Yaskawa INFORM job: R1_W27-A5(90,0)OK-KM.JBI

/JOB
//NAME R1_W27-A5(90,0)OK-KM
///FOLDERNAME KRIS-SCIANA
//POS
///NPOS 185,185,0,11,0,0
///TOOL 0
///POSTYPE PULSE
///PULSE
C00000=37728,-25402,-59646,12123,81500,-87547
C00001=37728,-25402,-59646,12123,81500,-87547
C00002=91138,-155068,-109614,11761,-43738,-37693
C00003=119745,-153431,-102899,11459,-45100,-35884
C00004=119745,-153431,-102899,-27163,23845,-36063
C00005=82911,-33235,-23976,-38303,40316,-52135
C00006=76873,-23146,-17071,-33335,38547,-55116
C00007=77767,-16866,-4062,-37722,34988,-52633
C00008=77963,-15290,-967,-38851,34204,-52007
C00009=77963,-14962,-89,-39196,33912,-51822
C00010=77963,-15290,-967,-38851,34204,-52007
C00011=74912,-28085,-18084,-33157,36163,-55249
C00012=87425,-27898,-13680,-43892,39692,-48702
C00013=86506,-25121,-9781,-44194,38523,-48572
C00014=85850,-24209,-8487,-44098,37958,-48664
C00015=86506,-25121,-9781,-44194,38523,-48572
C00016=88499,-29485,-18641,-42732,41870,-49349
C00017=84065,-39934,-28269,-47565,31902,-47281
C00018=97660,-57598,-46315,-76057,51112,-44177
C00019=97660,-57598,-46315,-76057,51112,22687
C00020=84258,-1988,-20698,-34156,82686,37449
C00021=71650,44734,31864,-29990,67100,37520
C00022=68559,51841,34481,-21650,72595,35300
C00023=68559,52177,36557,-21773,71566,35494
C00024=71650,44734,31864,-29990,67100,37520
C00025=70945,44192,31290,-29757,66915,37278
C00026=71650,44734,31864,-29990,67100,37520
C00027=73638,27072,10407,-29859,71409,37151
C00028=84818,-5861,-34609,-25685,107970,66305
C00029=82304,-18126,-38436,-25115,103648,66333
C00030=82304,-18241,-37568,-25043,103108,66450
C00031=82304,-18126,-38436,-25115,103648,66333
C00032=81928,-19595,-39516,-25102,103455,66234
C00033=82304,-18126,-38436,-25115,103648,66333
C00034=89590,-10169,-38886,-25731,109749,67700
C00035=79821,25746,-12201,-14172,109985,-51685
C00036=75346,32608,-5411,-14115,108620,-53087
C00037=69367,42381,13672,-2650,109038,-53623
C00038=69672,41657,12911,-2619,109144,-53518
C00039=69367,42407,13451,-2654,109187,-53626
C00040=69778,41548,11559,-2621,109922,-53494
C00041=69778,41458,12200,-2614,109483,-53485
C00042=69778,41717,10519,-2636,110650,-53511
C00043=75546,32003,-7767,-2128,117063,-51505
C00044=89590,-10367,-38270,-25645,109314,67802
C00045=81318,-16645,-42899,-25578,106543,65314
C00046=81011,-17824,-43775,-25562,106392,65231
C00047=81318,-16645,-42899,-25578,106543,65314
C00048=81318,-16217,-44241,-25738,107491,65096
C00049=80508,-19487,-45963,-25627,106690,64976
C00050=80508,-19653,-45420,-25564,106310,65064
C00051=80508,-19487,-45963,-25627,106690,64976
C00052=95846,-36399,-54281,-36372,102338,70376
C00053=102769,-67405,-57032,-50388,80798,81585
C00054=102006,-67104,-56883,-50326,80418,81392
C00055=101071,-66717,-56691,-50243,79954,81156
C00056=102358,-67245,-56953,-50356,80595,81483
C00057=109446,-46040,-50390,-50619,88983,80633
C00058=76818,2269,-30427,-25766,107073,87842
C00059=74377,-18,-31232,-25562,105749,87240
C00060=73964,56,-31169,-25544,105627,87112
C00061=74377,-18,-31232,-25562,105749,87240
C00062=74377,525,-32636,-25731,106781,87003
C00063=73295,1251,-31494,-25627,106170,86744
C00064=73295,967,-30757,-25541,105628,86868
C00065=73295,1251,-31494,-25627,106170,86744
C00066=70279,40415,5647,-25108,102815,86384
C00067=70279,40232,6317,-25050,102354,86487
C00068=70279,40415,5647,-25108,102815,86384
C00069=71244,41386,6665,-25146,102979,86705
C00070=70901,41880,8462,-25047,102103,86769
C00071=70442,41953,8538,-25022,101961,86631
C00072=70902,41930,8262,-25048,102238,86740
C00073=61610,48110,15922,-22399,84700,84261
C00074=61413,48286,16169,-22315,84306,84210
C00075=61008,48239,16118,-22214,84206,84086
C00076=61413,48286,16169,-22315,84306,84210
C00077=61413,48513,15025,-22296,85069,84067
C00078=60697,48720,15417,-22121,84760,83876
C00079=60697,48582,16098,-22134,84306,83960
C00080=60697,48720,15417,-22121,84760,83876
C00081=63518,20060,-6225,-30680,67231,85063
C00082=64098,14214,-10771,-32409,63712,85286
C00083=68885,5587,-7565,-48592,41009,78461
C00084=65627,18359,4931,-47317,38515,77893
C00085=65380,18933,5464,-47167,38362,77820
C00086=65627,18359,4931,-47317,38515,77893
C00087=65627,18423,5468,-47595,38308,78054
C00088=65627,18359,4931,-47317,38515,77893
C00089=70388,-714,-11888,-50078,41438,79261
C00090=70090,148,-11169,-50028,41395,-62740
C00091=64431,-8095,-22559,-54079,48047,-56053
C00092=60138,2499,-10245,-53390,44291,-56175
C00093=60864,4119,-8811,-53841,44675,-55941
C00094=50454,6570,-14378,-8272,39887,-77071
C00095=46890,10124,-11410,8335,39857,-85304
C00096=49558,3708,-17404,-7293,40191,-77557
C00097=52170,-20958,-36880,-10077,39785,-76177
C00098=53236,-23702,-38850,-11204,39728,-75616
C00099=68411,-25809,-57189,-29389,70593,82687
C00100=64998,-21965,-41730,-29205,62846,83456
C00101=47332,3816,-28668,-14363,85152,86760
C00102=13605,-12882,-44436,-5505,92305,85655
C00103=22082,-48383,-67711,-6096,86634,88967
C00104=44284,-41688,-65263,-13455,83816,85908
C00105=48658,1110,-32244,-14746,86156,87078
C00106=44206,2405,-29873,-10094,85398,89089
C00107=46271,27497,-4271,-10640,75407,89194
C00108=49813,9574,-21485,-13963,73922,89293
C00109=51221,-59455,-73476,-13519,71647,80934
C00110=20614,-34885,-59650,-13331,96803,87930
C00111=10167,-61122,-75524,-13198,98224,81006
C00112=18568,-72268,-87151,-10294,92386,67226
C00113=26792,-77751,-90608,-11605,92779,-33394
C00114=45042,-57080,-44270,-29328,87501,-26999
C00115=29931,-98809,-62657,-30113,73342,-29188
C00116=11116,-94328,-56612,-18416,63270,-35426
C00117=11737,-97137,-54513,-22781,52265,-32783
C00118=45210,-102279,-54102,-43605,63453,-17867
C00119=65059,-108164,-59991,-34964,63220,70148
C00120=52273,-70600,-39377,-24696,79942,57751
C00121=43673,-95736,-42893,-26460,67675,57325
C00122=28563,-66776,-31973,-25457,70564,50966
C00123=34229,-67024,-36548,-25195,74692,52186
C00124=29998,-46574,-23957,-5282,52394,19779
C00125=26910,-15086,7402,-4123,49104,18623
C00126=30725,5348,23556,-5801,49891,20233
C00127=26399,10546,29797,6839,45413,17161
C00128=25240,116,19359,9501,43500,14765
C00129=22231,-28513,-5139,11190,44238,13411
C00130=78144,-23782,-17517,-19802,53604,-33534
C00131=71297,46402,29834,-2695,101694,-44274
C00132=54466,25430,16217,2924,106693,-49878
C00133=60216,41298,32233,4120,104740,-47883
C00134=58235,32090,17782,3799,108986,-48454
C00135=79593,-22722,-23344,-19568,57852,-33734
C00136=78528,-18616,-11242,-20296,52560,-33151
C00137=78932,-16743,-10167,-20417,52946,-33052
C00138=78544,-16737,-8595,-20480,51941,-33014
C00139=77955,-18452,-11115,-20012,52425,-33380
C00140=78575,-16130,-9486,-20269,52757,-33170
C00141=76564,-15411,-8500,-18566,50879,-33728
C00142=75844,-13833,-7410,-18312,50740,-34021
C00143=76952,-15561,-8970,-19469,52340,-33810
C00144=76532,-19770,-12086,-19320,52008,-33932
C00145=90733,-10813,-5342,-38854,64320,-29793
C00146=90042,-7330,-2603,-38655,64092,-30029
C00147=89654,-5763,-1731,-38480,64131,-30226
C00148=90645,-6898,-2268,-38798,64375,-29857
C00149=90264,-6063,-535,-38894,63701,-29768
C00150=89843,-4938,-962,-38544,64174,-30154
C00151=90707,-2014,1381,-38736,64612,-29923
C00152=91454,1636,4460,-38922,64932,-29697
C00153=91128,-2551,1262,-38897,64640,-29735
C00154=91822,-6037,-1569,-39075,64914,-29517
C00155=89351,12292,-5617,-20131,79037,60764
C00156=89352,16382,17787,-21350,67492,62811
C00157=87694,16715,18095,-20947,67047,62250
C00158=87033,16875,18243,-20783,66871,62026
C00159=87546,18694,19932,-20926,66903,62219
C00160=87127,16733,16861,-20697,67624,61924
C00161=86853,17243,18585,-20744,66809,61967
C00162=87778,19395,20596,-20991,66917,62307
C00163=93870,634,-11523,-21410,77965,27109
C00164=93832,30424,31287,-31485,89224,-4964
C00165=93834,30423,31286,-31485,89224,-4963
C00166=93835,30423,31286,-31485,89225,-4963
C00167=93885,30318,29928,-31492,89915,-5134
C00168=93558,28166,29049,-31504,89308,-5095
C00169=93835,30423,31286,-31484,89222,-4963
C00170=93835,30427,31290,-31485,89224,-4963
C00171=93832,30428,31291,-31485,89223,-4964
C00172=78422,20921,22036,-838,76825,9185
C00173=78437,23453,23148,-839,77442,9187
C00174=77317,26936,27718,2138,78128,8741
C00175=79840,22908,23920,-1007,76703,9676
C00176=79114,23558,23278,-919,77424,9420
C00177=78338,19571,8789,758,86105,8103
C00178=114533,-1412,-14551,-12904,94461,10066
C00179=113047,-133639,-110380,-13907,-12366,10665
C00180=113047,-161651,-128625,-13333,-12898,10403
C00181=3699,-161651,-128625,-13333,-12898,10403
C00182=3699,-161651,-128625,-13333,-12898,-84221
C00183=-5596,-96163,-97527,-5645,15530,-80546
C00184=-5408,65526,-18493,9932,83824,-70089
BC00000=244758,1245750,1068204
BC00001=244758,1188259,1068204
BC00002=328514,1188626,1057284
BC00003=25914,1188837,1050998
BC00004=25914,1188837,250553
BC00005=876,1188837,301895
BC00006=876,1188837,280170
BC00007=876,1188837,280170
BC00008=876,1188837,280170
BC00009=876,1188837,280170
BC00010=876,1188837,280170
BC00011=876,1188837,280170
BC00012=876,1188837,280170
BC00013=876,1188837,280170
BC00014=876,1188837,280170
BC00015=876,1188837,280170
BC00016=876,1188837,280170
BC00017=876,1188837,242031
BC00018=876,1188837,199876
BC00019=876,1188837,199876
BC00020=876,1188837,199876
BC00021=876,1188837,199876
BC00022=876,1188837,199876
BC00023=876,1188837,199876
BC00024=876,1188837,199876
BC00025=876,1188837,199873
BC00026=876,1188837,199876
BC00027=876,1188837,199876
BC00028=876,1188837,199876
BC00029=876,1188837,199876
BC00030=876,1188837,199876
BC00031=876,1188837,199876
BC00032=876,1188837,199876
BC00033=876,1188837,199876
BC00034=876,1188837,199876
BC00035=876,1188837,199876
BC00036=876,1188837,199876
BC00037=876,1188837,199876
BC00038=876,1188837,199876
BC00039=876,1188837,199876
BC00040=876,1188837,199876
BC00041=876,1188837,199876
BC00042=876,1188837,199876
BC00043=876,1188837,200133
BC00044=876,1188837,583866
BC00045=876,1188837,583866
BC00046=876,1188837,583866
BC00047=876,1188837,583866
BC00048=876,1188837,583866
BC00049=876,1188837,583866
BC00050=876,1188837,583866
BC00051=876,1188837,583866
BC00052=876,1188837,583866
BC00053=876,1188837,597308
BC00054=876,1188837,597308
BC00055=876,1188837,597308
BC00056=876,1188837,597308
BC00057=876,1188837,597308
BC00058=876,1188837,587630
BC00059=876,1188837,587630
BC00060=876,1188837,587630
BC00061=876,1188837,587630
BC00062=876,1188837,587630
BC00063=876,1188837,587630
BC00064=876,1188837,587630
BC00065=876,1188837,587630
BC00066=876,1188837,587630
BC00067=876,1188837,587630
BC00068=876,1188837,587630
BC00069=876,1188837,587630
BC00070=876,1188837,587628
BC00071=876,1188837,587628
BC00072=876,1188837,587630
BC00073=876,1156999,587630
BC00074=876,1156326,587630
BC00075=876,1156326,587630
BC00076=876,1156326,587630
BC00077=876,1156326,587630
BC00078=876,1156326,587630
BC00079=876,1156326,587630
BC00080=876,1156326,587630
BC00081=876,1156326,587630
BC00082=876,1156326,597308
BC00083=876,1156326,697181
BC00084=876,1156326,697181
BC00085=876,1156326,697181
BC00086=876,1156326,697181
BC00087=876,1156326,697181
BC00088=876,1156326,697181
BC00089=876,1156326,697181
BC00090=876,1156326,697181
BC00091=876,1128921,697181
BC00092=876,1128921,697181
BC00093=876,1128921,697181
BC00094=876,1128921,697181
BC00095=876,1128922,697179
BC00096=876,1128921,697181
BC00097=876,1128921,697181
BC00098=876,1128921,697181
BC00099=1315,1138846,645939
BC00100=1315,1138846,645939
BC00101=1732,1122257,597308
BC00102=2782,1039755,587713
BC00103=2792,1082515,587630
BC00104=1732,1122257,587630
BC00105=1732,1122257,587630
BC00106=1732,1122257,587630
BC00107=1732,1122257,587630
BC00108=1732,1122257,587630
BC00109=1732,1122257,587630
BC00110=1732,1065745,587630
BC00111=1732,1065745,587630
BC00112=1732,1065745,587630
BC00113=1732,1065745,597308
BC00114=1732,1065745,805135
BC00115=1732,1066766,805135
BC00116=1732,1066766,791693
BC00117=1732,1066766,791693
BC00118=1732,1066766,805135
BC00119=1732,1066766,805135
BC00120=1732,1066766,417253
BC00121=29114,1066766,417253
BC00122=5096,1066766,417253
BC00123=1732,1066766,417253
BC00124=1732,1066766,417253
BC00125=1732,1066766,417253
BC00126=1732,1066766,417253
BC00127=1732,1066766,417253
BC00128=1732,1066766,417253
BC00129=1732,1066766,417253
BC00130=876,1188837,310651
BC00131=876,1188837,310651
BC00132=876,1149728,310651
BC00133=876,1149728,310651
BC00134=876,1149728,310651
BC00135=876,1384690,305516
BC00136=876,1384690,305516
BC00137=876,1384690,297010
BC00138=876,1384690,297010
BC00139=876,1384690,297010
BC00140=876,1384690,297005
BC00141=876,1384690,296893
BC00142=876,1384690,296887
BC00143=876,1384690,305393
BC00144=876,1384690,326658
BC00145=876,1384690,316977
BC00146=876,1384690,294261
BC00147=876,1384690,285175
BC00148=876,1384690,285175
BC00149=876,1384690,285175
BC00150=876,1384690,285189
BC00151=876,1384690,285231
BC00152=876,1384690,285245
BC00153=876,1384690,294331
BC00154=876,1384690,317047
BC00155=876,1384690,372171
BC00156=876,1384690,372171
BC00157=876,1384690,350251
BC00158=876,1384690,341483
BC00159=876,1384690,341483
BC00160=876,1384690,341483
BC00161=876,1384690,341468
BC00162=876,1384690,372038
BC00163=876,1384690,372038
BC00164=6218,1373517,366370
BC00165=10148,1372468,343278
BC00166=11720,1372049,334041
BC00167=11720,1372049,334041
BC00168=11720,1372049,334041
BC00169=12357,1372055,334027
BC00170=15563,1372482,343131
BC00171=11633,1373530,366223
BC00172=7822,1384690,403141
BC00173=10818,1384690,380007
BC00174=12016,1384690,370753
BC00175=12016,1384690,370753
BC00176=12016,1384690,370753
BC00177=10869,1187534,355175
BC00178=877,1178820,383119
BC00179=877,1178820,1012132
BC00180=877,1178820,1012132
BC00181=125475,1178820,1012132
BC00182=354926,1178820,1012132
BC00183=329290,1178681,1025649
BC00184=165568,1305468,1058537
///POSTYPE BASE
///RECTAN
///RCONF 0,0,0,0,0,0,0,0,0,0,0,0,0,0,0,0,0,0,0,0,0,0,0,0
P00006=0.222,-3.123,-1.508,0.0000,0.0000,0.0000
P00022=0.222,-3.123,-1.508,0.0000,0.0000,0.0000
P00023=0.143,-0.036,0.682,0.0000,0.0000,0.0000
P00024=0.145,-0.552,1.326,0.0000,0.0000,0.0000
P00025=-2.003,0.006,0.728,0.0000,0.0000,0.0000
P00026=0.562,-0.002,-0.337,0.0000,0.0000,0.0000
P00027=-0.746,0.015,-9.096,0.0000,0.0000,0.0000
P00028=-2.237,-0.018,-7.702,0.0000,0.0000,0.0000
P00029=-2.156,-0.086,-4.681,0.0000,0.0000,0.0000
P00030=5.926,-4.294,-1.390,0.0000,0.0000,0.0000
P00035=2.817,0.591,-1.622,0.0000,0.0000,0.0000
//INST
///DATE 2024/07/29 21:04
///ATTR SC,RW
///GROUP1 RB1,BS1
NOP
SFTOF
MOVJ C00000 BC00000 VJ=50.00
MOVJ C00001 BC00001 VJ=100.00
MOVJ C00002 BC00002 VJ=100.00
MOVJ C00003 BC00003 VJ=100.00
MOVJ C00004 BC00004 VJ=100.00
MOVL C00005 BC00005 V=166.7
MOVL C00006 BC00006 V=166.7
MOVL C00007 BC00007 V=100.0
MOVL C00008 BC00008 V=60.0
REFP 3 C00009 BC00009
CALL JOB:SEARCH-R1
SET P028 P006
SFTON P028
MOVL C00010 BC00010 V=60.0
MOVL C00011 BC00011 V=133.3
MOVL C00012 BC00012 V=133.3
MOVL C00013 BC00013 V=60.0
REFP 3 C00014 BC00014
CALL JOB:SEARCH-R1
SET P028 P006
SFTON P028
MOVL C00015 BC00015 V=60.0
MOVL C00016 BC00016 V=133.3
MOVL C00017 BC00017 V=166.7
'Path S1011
SFTOF
'Path VIA1114
SFTOF
MOVJ C00018 BC00018 VJ=100.00
MOVJ C00019 BC00019 VJ=100.00
'POMIAR NOWE SPOINY
MOVJ C00020 BC00020 VJ=100.00
MOVJ C00021 BC00021 VJ=15.00
MOVL C00022 BC00022 V=83.3
REFP 3 C00023 BC00023
CALL JOB:SEARCH-R1
SET P022 P006
SFTON P022
MOVL C00024 BC00024 V=60.0
REFP 3 C00025 BC00025
CALL JOB:SEARCH-R1
SET P022 P006
SFTON P022
MOVL C00026 BC00026 V=60.0
SFTOF
MOVL C00027 BC00027 V=83.3
MOVL C00028 BC00028 V=83.3
MOVL C00029 BC00029 V=166.7
REFP 3 C00030 BC00030
CALL JOB:SEARCH-R1
SET P023 P006
SFTON P023
MOVL C00031 BC00031 V=60.0
REFP 3 C00032 BC00032
CALL JOB:SEARCH-R1
SET P023 P006
SFTON P023
MOVL C00033 BC00033 V=60.0
MOVJ C00034 BC00034 VJ=15.00
MOVJ C00035 BC00035 VJ=15.00
SFTOF
MOVJ C00036 BC00036 VJ=15.00
'POPRAWIC POMIAR
MOVJ C00037 BC00037 VJ=15.00
REFP 3 C00038 BC00038
CALL JOB:SEARCH-R1
SET P030 P006
SFTON P030
MOVL C00039 BC00039 V=60.0
MOVL C00040 BC00040 V=166.7
REFP 3 C00041 BC00041
CALL JOB:SEARCH-R1
SET P030 P006
SFTON P030
MOVL C00042 BC00042 V=100.0
MOVJ C00043 BC00043 VJ=15.00
SFTOF
MOVJ C00044 BC00044 VJ=50.00
MOVJ C00045 BC00045 VJ=15.00
REFP 3 C00046 BC00046
CALL JOB:SEARCH-R1
SET P024 P006
SFTON P024
MOVL C00047 BC00047 V=60.0
MOVL C00048 BC00048 V=166.7
MOVL C00049 BC00049 V=166.7
REFP 3 C00050 BC00050
CALL JOB:SEARCH-R1
SET P024 P006
SFTON P024
MOVL C00051 BC00051 V=60.0
MOVJ C00052 BC00052 VJ=15.00
SFTOF
MOVJ C00053 BC00053 VJ=15.00
MOVL C00054 BC00054 V=83.3
REFP 3 C00055 BC00055
CALL JOB:SEARCH-R1
SET P024 P006
SFTON P024
MOVL C00056 BC00056 V=83.3
MOVL C00057 BC00057 V=833.3
MOVJ C00058 BC00058 VJ=15.00
MOVL C00059 BC00059 V=100.0
REFP 3 C00060 BC00060
CALL JOB:SEARCH-R1
SET P025 P006
SFTON P025
MOVL C00061 BC00061 V=100.0
MOVL C00062 BC00062 V=166.7
MOVL C00063 BC00063 V=166.7
REFP 3 C00064 BC00064
CALL JOB:SEARCH-R1
SET P025 P006
SFTON P025
MOVL C00065 BC00065 V=60.0
SFTOF
MOVL C00066 BC00066 V=166.7
REFP 3 C00067 BC00067
CALL JOB:SEARCH-R1
SET P026 P006
SFTON P026
MOVL C00068 BC00068 V=60.0
MOVL C00069 BC00069 V=166.7
MOVL C00070 BC00070 V=166.7
REFP 3 C00071 BC00071
CALL JOB:SEARCH-R1
SET P026 P006
SFTON P026
MOVL C00072 BC00072 V=100.0
SFTOF
MOVL C00073 BC00073 V=300.0
MOVL C00074 BC00074 V=166.7
REFP 3 C00075 BC00075
CALL JOB:SEARCH-R1
SET P027 P006
SFTON P027
MOVL C00076 BC00076 V=166.7
MOVL C00077 BC00077 V=166.7
MOVL C00078 BC00078 V=166.7
REFP 3 C00079 BC00079
CALL JOB:SEARCH-R1
SET P027 P006
SFTON P027
MOVL C00080 BC00080 V=250.0
SFTOF
MOVL C00081 BC00081 V=166.7
MOVJ C00082 BC00082 VJ=15.00
MOVJ C00083 BC00083 VJ=30.00
MOVJ C00084 BC00084 VJ=15.00
REFP 3 C00085 BC00085
CALL JOB:SEARCH-R1
SET P035 P006
SFTON P035
MOVL C00086 BC00086 V=60.0
REFP 3 C00087 BC00087
CALL JOB:SEARCH-R1
SET P035 P006
SFTON P035
MOVL C00088 BC00088 V=60.0
SFTOF
MOVJ C00089 BC00089 VJ=15.00
MOVJ C00090 BC00090 VJ=15.00
MOVL C00091 BC00091 V=50.0
MACRO1 MJ#(0) ARGF7
SFTON P035
MOVL C00092 BC00092 V=50.0
ARCON
MOVL C00093 BC00093 V=7.5
MOVL C00094 BC00094 V=7.5
MOVL C00095 BC00095 V=7.5
ARCOF
SFTOF
MOVL C00096 BC00096 V=25.0
MOVL C00097 BC00097 V=66.7
MOVJ C00098 BC00098 VJ=15.00
MOVJ C00099 BC00099 VJ=15.00
MOVJ C00100 BC00100 VJ=15.00
MACRO1 MJ#(0) ARGF7
MOVL C00101 BC00101 V=166.7
SFTON P027
MOVL C00102 BC00102 V=166.7
ARCON
MOVL C00103 BC00103 V=11.7
ARCOF
SFTOF
MOVJ C00104 BC00104 VJ=15.00
MOVJ C00105 BC00105 VJ=15.00
SFTON P027
MOVJ C00106 BC00106 VJ=15.00
ARCON
MOVL C00107 BC00107 V=11.7
ARCOF
SFTOF
MOVJ C00108 BC00108 VJ=15.00
MOVJ C00109 BC00109 VJ=15.00
SFTON P026
MOVJ C00110 BC00110 VJ=15.00
ARCON
SFTON P025
MOVL C00111 BC00111 V=11.7
ARCOF
SFTOF
MOVJ C00112 BC00112 VJ=15.00
MOVJ C00113 BC00113 VJ=15.00
MOVJ C00114 BC00114 VJ=15.00
MACRO1 MJ#(0) ARGF12
MOVJ C00115 BC00115 VJ=15.00
SFTON P024
MOVJ C00116 BC00116 VJ=15.00
ARCON
MOVL C00117 BC00117 V=12.5
ARCOF
SFTOF
MOVJ C00118 BC00118 VJ=15.00
MOVJ C00119 BC00119 VJ=15.00
MACRO1 MJ#(0) ARGF6
MOVJ C00120 BC00120 VJ=15.00
SFTON P023
MOVJ C00121 BC00121 VJ=15.00
ARCON
MOVL C00122 BC00122 V=9.2
ARCOF
MOVJ C00123 BC00123 VJ=15.00
SFTOF
MOVJ C00124 BC00124 VJ=15.00
SFTON P022
MOVJ C00125 BC00125 VJ=15.00
ARCON
MOVL C00126 BC00126 V=7.5
MOVL C00127 BC00127 V=7.5
ARCOF
SFTOF
MOVJ C00128 BC00128 VJ=15.00
MOVJ C00129 BC00129 VJ=15.00
MOVL C00130 BC00130 V=166.7
MACRO1 MJ#(0) ARGF6
MOVL C00131 BC00131 V=83.3
SFTON P030
'POPRAWIC POMIAR
MOVL C00132 BC00132 V=83.3
ARCON
MOVL C00133 BC00133 V=7.5
ARCOF
SFTOF
MOVJ C00134 BC00134 VJ=15.00
COMM MACRO1 MJ#(0) ARGF7
COMM MOVL C00135 BC00135 V=166.7
COMM MOVL C00136 BC00136 V=166.7
COMM SFTON P028
COMM MOVL C00137 BC00137 V=100.0 PL=0
COMM REFP 1 C00138 BC00138
COMM REFP 2 C00139 BC00139
COMM MACRO1 MJ#(0) ARGF7
COMM MOVL C00140 BC00140 V=10.0
COMM MOVL C00141 BC00141 V=10.0
COMM MOVL C00142 BC00142 V=10.0
COMM ARCOF
COMM MOVL C00143 BC00143 V=166.7
COMM MOVL C00144 BC00144 V=166.7
COMM SFTOF
COMM 'Path W1013
COMM SFTOF
COMM SFTON P028
COMM MOVL C00145 BC00145 V=166.7
COMM MOVL C00146 BC00146 V=166.7
COMM MOVL C00147 BC00147 V=100.0 PL=0
COMM REFP 1 C00148 BC00148
COMM REFP 2 C00149 BC00149
COMM MACRO1 MJ#(0) ARGF7
COMM MOVL C00150 BC00150 V=10.0
COMM MOVL C00151 BC00151 V=10.0
COMM MOVL C00152 BC00152 V=10.0
COMM ARCOF
COMM MOVL C00153 BC00153 V=166.7
COMM MOVL C00154 BC00154 V=166.7
COMM SFTOF
COMM 'Path VIA1116
COMM SFTOF
COMM MOVJ C00155 BC00155 VJ=100.00
COMM 'Path W1014
COMM SFTOF
COMM SFTON P028
COMM MOVL C00156 BC00156 V=166.7
COMM MOVL C00157 BC00157 V=166.7
COMM 'NIE SPAWAMY-BRAK MIEJSCA
COMM MOVL C00158 BC00158 V=100.0 PL=0
COMM REFP 1 C00159 BC00159
COMM REFP 2 C00160 BC00160
COMM MACRO1 MJ#(0) ARGF7
COMM MOVL C00161 BC00161 V=10.0
COMM ARCOF
COMM MOVL C00162 BC00162 V=166.7
COMM SFTOF
COMM 'Path VIA1117
COMM SFTOF
COMM MOVJ C00163 BC00163 VJ=100.00
COMM 'Path W1015
COMM SFTOF
COMM SFTON P029
COMM MOVL C00164 BC00164 V=1000.0
COMM MOVL C00165 BC00165 V=400.0
COMM MOVL C00166 BC00166 V=100.0 PL=0
COMM REFP 1 C00167 BC00167
COMM REFP 2 C00168 BC00168
COMM MACRO1 MJ#(0) ARGF0
COMM MOVL C00169 BC00169 V=10.0
COMM ARCOF
COMM MOVL C00170 BC00170 V=400.0
COMM MOVL C00171 BC00171 V=166.7
COMM SFTOF
COMM 'Path W1016
COMM SFTOF
COMM SFTON P029
COMM MOVL C00172 BC00172 V=166.7
COMM MOVL C00173 BC00173 V=166.7
COMM MOVL C00174 BC00174 V=100.0 PL=0
COMM REFP 1 C00175 BC00175
COMM REFP 2 C00176 BC00176
COMM MACRO1 MJ#(0) ARGF7
COMM ARCOF
MOVL C00177 BC00177 V=166.7
SFTOF
MOVJ C00178 BC00178 VJ=100.00
MOVJ C00179 BC00179 VJ=100.00
MOVJ C00180 BC00180 VJ=100.00
MOVJ C00181 BC00181 VJ=100.00
MOVJ C00182 BC00182 VJ=100.00
MOVJ C00183 BC00183 VJ=100.00
MOVJ C00184 BC00184 VJ=40.00
END
